Staubli VAL3: _startSimul.pgx

program _startSimul(InstrItem& x_iInstr (dimensions=1))
  local bool l_bContinue
  local string l_sEvent
begin
  // init all
  call cycleStatus:init()
  // CHECK FOR CYCLE EVENT
  if !cycleStatus:bCycle and !cycleStatus:bSimulation
    // set the Simulation is ON
    cycleStatus:bSimulation=true
    if x_iInstr.sType=="HOME"
      cycleStatus:bHoming=true
    endIf
    // SIMULATION
    logMsg("[KERNEL] SUPERVISOR:Interface>Simulation of the event: "+x_iInstr.sType+" "+x_iInstr.sData)
    taskCreate "Simulation",50,cycle_simul(x_iInstr)
    // start the action Task for the traj
    taskCreate "Action",80,action_buffer()
  endIf
end
